(* CODESYS project GlobalConstants.export

Project tree, tasks and I/O mapping:
  GlobalConstants/
    Inficon/
      CommandID/
        global variables InficonHCommandID
        global variables InficonQCCommandID
        global variables InficonQGCommandID
        global variables InficonQMCommandID
        global variables InficonQSCommandID
        global variables InficonRGCommandID
        global variables InficonRLCommandID
        global variables InficonSGCommandID
        global variables InficonSLCommandID
        global variables InficonSSCommandID
      global variables InficonCommand
      global variables InficonQUSubgroup
      global variables InficonResponceErrorCode
      global variables InficonRSSubgroup
    global variables Constants
    global variables IPS_COMMAND
*)

// GlobalConstants/Constants
{attribute 'qualified_only'}
//{attribute 'conditionalshow'}
//{attribute 'conditionalshow' := 'SomeText'}
//{attribute 'hide'}
VAR_GLOBAL CONSTANT
	gc_iDummy : INT := 42; /// This is a dummy global constant variable
END_VAR

// GlobalConstants/IPS_COMMAND
{attribute 'qualified_only'}
VAR_GLOBAL CONSTANT
	START_PERMIT:	UINT:=101;
	START:			UINT:=1;
	STOP:			UINT:=2;
	RESET_ERROR:	UINT:=3;
	
END_VAR

// GlobalConstants/Inficon/InficonCommand
{attribute 'qualified_only'}
(*Основные командные группы.
Команда формируется по следующему шаблону COMMAND_GROUP[SUB GROUP][COMMAND ID](Parameter...Parameter)*)
VAR_GLOBAL CONSTANT
	Hello:BYTE:=STRING_TO_BYTE('H');
	Query:BYTE:=STRING_TO_BYTE('Q');
	RemoteAction:BYTE:=STRING_TO_BYTE('R');
	Status:BYTE:=STRING_TO_BYTE('S');
	Update:BYTE:=STRING_TO_BYTE('U');
	
END_VAR

// GlobalConstants/Inficon/InficonQUSubgroup
{attribute 'qualified_only'}
(*Subcommand for command 'Query' and 'Update's*)
VAR_GLOBAL CONSTANT
	Source:			BYTE:=STRING_TO_BYTE('C');
	General:		BYTE:=STRING_TO_BYTE('G');
	InputName: 		BYTE:=STRING_TO_BYTE('I');
	Logic:			BYTE:=STRING_TO_BYTE('L');
	Material:		BYTE:=STRING_TO_BYTE('M');
	MaterialName:	BYTE:=STRING_TO_BYTE('N');
	OutputName:		BYTE:=STRING_TO_BYTE('O');
	Process:		BYTE:=STRING_TO_BYTE('P');
	Sensor:			BYTE:=STRING_TO_BYTE('S');
	TypeOfOutput:	BYTE:=STRING_TO_BYTE('T');
	UserMessage:	BYTE:=STRING_TO_BYTE('V');
END_VAR

// GlobalConstants/Inficon/InficonResponceErrorCode
{attribute 'qualified_only'}
VAR_GLOBAL CONSTANT
	IllegalCommand:					BYTE:=STRING_TO_BYTE('A');
	IllegalParametervalue:			BYTE:=STRING_TO_BYTE('B');
	InvalidChecksum:				BYTE:=STRING_TO_BYTE('C');
	IllegalID:						BYTE:=STRING_TO_BYTE('D');
	DataNotAvailable:				BYTE:=STRING_TO_BYTE('E');
	IllegalFormat:					BYTE:=STRING_TO_BYTE('F');
	CannotDoNow:					BYTE:=STRING_TO_BYTE('F');
	InvalidMessage:					BYTE:=STRING_TO_BYTE('I');
	LengthError:					BYTE:=STRING_TO_BYTE('L');
	TooManyCommands:				BYTE:=STRING_TO_BYTE('M');
	ResponceLengthLarge:			BYTE:=STRING_TO_BYTE('O');
	ProiorCommandFailed:			BYTE:=STRING_TO_BYTE('P');
END_VAR

// GlobalConstants/Inficon/InficonRSSubgroup
{attribute 'qualified_only'}
VAR_GLOBAL CONSTANT
	General:	BYTE:=STRING_TO_BYTE('G');
 	Material:	BYTE:=STRING_TO_BYTE('L');
	Sensor:		BYTE:=STRING_TO_BYTE('S');
END_VAR

// GlobalConstants/Inficon/CommandID/InficonHCommandID
{attribute 'qualified_only'}
VAR_GLOBAL
	NameAndVersion: 	BYTE:=16#01;
	VersionNumbers:		BYTE:=16#02;
	FirmawareVersion: 	BYTE:=16#03;
END_VAR

// GlobalConstants/Inficon/CommandID/InficonQCCommandID
{attribute 'qualified_only'}
VAR_GLOBAL CONSTANT
	DACOutput: 			BYTE:=16#01;
	ShutterOutput:		BYTE:=16#02;
	NumberOfCrucibles:	BYTE:=16#03;
	CrucibleOutput:		BYTE:=16#04;
	TurretFeedback:		BYTE:=16#05;
	TurretInput:		BYTE:=16#06;
	TurretDelay:		BYTE:=16#07;
END_VAR

// GlobalConstants/Inficon/CommandID/InficonQGCommandID
{attribute 'qualified_only'}
VAR_GLOBAL CONSTANT
	ThinknessEq1:		BYTE:=16#09;
	ThinknessEq2:		BYTE:=16#0A;
	ThinknessEq3:		BYTE:=16#0B;
	Test:				BYTE:=16#0C;
	TimeCompressed:		BYTE:=16#0D;//10x time acceleration
	AdvancedTest:		BYTE:=16#0E;//Crystal Fails Active
	AudioFeedback:		BYTE:=16#0F;
	LCDDimmerTime:		BYTE:=16#10;
	DateFormat:			BYTE:=16#11;
	USBDatalogFormat:	BYTE:=16#12;
	DatalogXtalInfo:	BYTE:=16#13;
	GraphScale:			BYTE:=16#14;
	GraphScaleRate:		BYTE:=16#15;
	RS232Baudrate:		BYTE:=16#16;
	RS232Protocol:		BYTE:=16#17;
	DAC1Scale:			BYTE:=16#18;
	DAC2Scale:			BYTE:=16#19;
	DAC3Scale:			BYTE:=16#1A;
	DAC4Scale:			BYTE:=16#1B;
	DAC5Scale:			BYTE:=16#1C;
	DAC6Scale:			BYTE:=16#1D;
	DAC7Scale:			BYTE:=16#1E;
	DAC8Scale:			BYTE:=16#1F;
	DAC9Scale:			BYTE:=16#20;
	DAC10Scale:			BYTE:=16#21;
	DAC11Scale:			BYTE:=16#22;
	DAC12Scale:			BYTE:=16#23;
	DAC1Polarity:		BYTE:=16#24;
	DAC2Polarity:		BYTE:=16#25;
	DAC3Polarity:		BYTE:=16#26;
	DAC4Polarity:		BYTE:=16#27;
	DAC5Polarity:		BYTE:=16#28;
	DAC6Polarity:		BYTE:=16#29;
	DAC7Polarity:		BYTE:=16#2A;
	DAC8Polarity:		BYTE:=16#2B;
	DAC9Polarity:		BYTE:=16#2C;
	DAC10Polarity:		BYTE:=16#2D;
	DAC11Polarity:		BYTE:=16#2E;
	DAC12Polarity:		BYTE:=16#2F;
	Channel1GraphScale:	BYTE:=16#31;
	Channel2GraphScale:	BYTE:=16#32;
	Channel3GraphScale:	BYTE:=16#33;
	Channel4GraphScale:	BYTE:=16#34;
	Channel5GraphScale:	BYTE:=16#35;
	Channel6GraphScale:	BYTE:=16#36;
	
	
END_VAR

// GlobalConstants/Inficon/CommandID/InficonQMCommandID
{attribute 'qualified_only'}
VAR_GLOBAL CONSTANT
	Density:			BYTE:=16#01;
	ZRation:			BYTE:=16#02;
	MasterTooling:		BYTE:=16#03;
	ControlLoop:		BYTE:=16#04;
	ProcessGain:		BYTE:=16#05;
	TimeConstant:		BYTE:=16#06;
	DeadTime:			BYTE:=16#07;
	MaximumPower:		BYTE:=16#09;
	MinimumPower:		BYTE:=16#0A;
	MaxPowerOption:		BYTE:=16#0B;
	PreCondSoakPower:	BYTE:=16#0C;
	PreCondRiseTime:	BYTE:=16#0D;
	PreCondSoakTime:	BYTE:=16#0E;
	SoakPower1:			BYTE:=16#0F;
	RiseTime1:			BYTE:=16#10;
	SoakTime1:			BYTE:=16#11;
	SoakPower2:			BYTE:=16#12;
	RiseTime2:			BYTE:=16#13;
	SoakTime:			BYTE:=16#14;
	AutoSoak2:			BYTE:=16#15;
	DepAfterPreDep:		BYTE:=16#16;
	DelayOption:		BYTE:=16#17;
	ControlDelayTime:	BYTE:=16#18;
	ShutterDelayAccur:	BYTE:=16#19;
	FeedPower:			BYTE:=16#1C;
	FeedRampTime:		BYTE:=16#1D;
	FeedTime:			BYTE:=16#1E;
	IdlePower:			BYTE:=16#20;
	Rate:				BYTE:=16#21;
	TimeLimit:			BYTE:=16#22;
	RateFilterTime:		BYTE:=16#23;
	TimePowerAvg:		BYTE:=16#24;
	IonAssitDeposite:	BYTE:=16#25;
	OnFinalThinckness:	BYTE:=16#26;
	Ramp1Rate:			BYTE:=16#27;
	StartRamp1:			BYTE:=16#28;
	Ramp1Time:			BYTE:=16#29;
	Ramp2Rate:			BYTE:=16#2A;
	StartRamp2:			BYTE:=16#2B;
	Ramp2Time:			BYTE:=16#2C;
	RateWatvherOption:	BYTE:=16#2D;
	RateWatcherTime:	BYTE:=16#2E;
	RateWatcherAccuracy:BYTE:=16#2F;
	FailureAction:		BYTE:=16#73;
	CrystalTwoTooling:	BYTE:=16#74;
	XtalPositionFirst:	BYTE:=16#75;
	XtalPositionLast:	BYTE:=16#76;
	QaulityPercent:		BYTE:=16#79;
	QualityCounts:		BYTE:=16#7A;
	StabilitySingle:	BYTE:=16#7B;
	StabilityTotal:		BYTE:=16#7C;
	RecorderOutput:		BYTE:=16#7D;
	RecorderFunction:	BYTE:=16#7E;
	RecorderRange:		BYTE:=16#7F;
	
	
	
END_VAR

// GlobalConstants/Inficon/CommandID/InficonQSCommandID
{attribute 'qualified_only'}
VAR_GLOBAL CONSTANT
	ShutterOut:			BYTE:=16#01;
	SensorType:			BYTE:=16#02;
	SitchOut:			BYTE:=16#03;
	AutoZ:				BYTE:=16#04;
	NumberOfPosition:	BYTE:=16#05;
	NumberOfPulse:		BYTE:=16#06;
	PulseOn:			BYTE:=16#07;
	PulseOff:			BYTE:=16#08;
	RecorderOutput:		BYTE:=16#09;
	RecorderFunction:	BYTE:=16#0A;
	RecorderRange:		BYTE:=16#0B;
	
END_VAR

// GlobalConstants/Inficon/CommandID/InficonRGCommandID
{attribute 'qualified_only'}
VAR_GLOBAL CONSTANT
	StopAll:						BYTE:=16#01;
	ResetAll:						BYTE:=16#02;
	RemoteLockOn:					BYTE:=16#03;
	RemoteLockOff:					BYTE:=16#04;
	SetLogicStatement:				BYTE:=16#05;
	ClearLogicStatement:			BYTE:=16#06;
	CrystalFailInhibitOn:			BYTE:=16#07;
	CrystalFailInhibitOff:			BYTE:=16#08;
	SetDate:						BYTE:=16#09;
	SetTime:						BYTE:=16#0A;
	ZeroCounter:					BYTE:=16#0B;
	ZeroTimer:						BYTE:=16#0C;
	StartTimer:						BYTE:=16#0D;
	ClockHoldOn:					BYTE:=16#0F;
	ClockHoldOff:					BYTE:=16#10;
	UserMessageOn:					BYTE:=16#11;
	UserMessageOff:					BYTE:=16#12;
	SoakHold1On:					BYTE:=16#13;
	SoakHold1Off:					BYTE:=16#14;
	SoakHold2On:					BYTE:=16#15;
	SoakHold2Off:					BYTE:=16#16;
	SwitchSensor:					BYTE:=16#17;
	ClearFailedCrystalsX:			BYTE:=16#18;
	RotateHeadX:					BYTE:=16#1A;
	DefaultAllParameters:			BYTE:=16#1B;
	SoakHoldPreConOn:				BYTE:=16#1D;
	SoakHoldPrecomOff:				BYTE:=16#1E;
	StartInhibitOn:					BYTE:=16#1F;
	StartIngibitOff:				BYTE:=16#20;
	RateWatcherSamplingInhibitOn:	BYTE:=16#21;
	RateWatcherSamplingInhibitOff:	BYTE:=16#22;
	WatcherSamplingInitiateOn:		BYTE:=16#23;
	WatcherSamplingInitiateOff:		BYTE:=16#24;
	ClearQAndSCountsForSensore:		BYTE:=16#25;
	NameMaterial:					BYTE:=16#26;
	
END_VAR

// GlobalConstants/Inficon/CommandID/InficonRLCommandID
{attribute 'qualified_only'}
VAR_GLOBAL CONSTANT
	StopMaterial:			BYTE:=16#00;
	ZeroThickness:			BYTE:=16#01;
	StartDeposit:			BYTE:=16#02;
	GoToNonDepositControl:	BYTE:=16#03;
	GoToPostDeposit:		BYTE:=16#04;
	ContinueDeposit:		BYTE:=16#05;
	GoToManual:				BYTE:=16#06;
	SetPowerlevel:			BYTE:=16#07;
	OpenSourceShutter:		BYTE:=16#08;
	CloseSourceShutter:		BYTE:=16#09;
	SetAverageRate:			BYTE:=16#0A;
	Start:					BYTE:=16#0B;
	ResetMaterial:			BYTE:=16#0C;
	
END_VAR

// GlobalConstants/Inficon/CommandID/InficonSGCommandID
{attribute 'qualified_only'}
VAR_GLOBAL CONSTANT
	OutputStatus: 				BYTE:=16#03; //Responce - 5 bytes. Каждый бит репрезентует OUTPUT
	InputStatus:				BYTE:=16#04; //Responce - 4 bytes
	LogicStatementStatus:		BYTE:=16#05; //Responce - 13 byte
	StatusMessage:				BYTE:=16#06; //Responce - 8 bytes
	StatusMessageDesignators:	BYTE:=16#07;
	TrancientMessages:			BYTE:=16#09; // Responce - 1 bytes
	SensorStatus:				BYTE:=16#0A;
	TimerStatus:				BYTE:=16#0B;
	TimerValue:					BYTE:=16#0C;
	CounterValue:				BYTE:=16#0D;
	ThicknessSum:				BYTE:=16#0E;
	GetDate:					BYTE:=16#0F;
	GetTime:					BYTE:=16#10;
	SystemConfuguration:		BYTE:=16#11;
	
	
END_VAR

// GlobalConstants/Inficon/CommandID/InficonSLCommandID
{attribute 'qualified_only'}
VAR_GLOBAL CONSTANT
	FilteredRate:			BYTE:=16#01;
	DisplayRate:			BYTE:=16#02;
	SourcePowerOutput:		BYTE:=16#03;
	Thickness:				BYTE:=16#04;
	State:					BYTE:=16#05;
	StateTime:				BYTE:=16#06;
	ActiveSensors:			BYTE:=16#07;
	PowerSourceNumber:		BYTE:=16#08;
	AccumulatedLayerTime:	BYTE:=16#09;
	DepositAverageRate:		BYTE:=16#0A;
	DepositAveragePower:	BYTE:=16#0B;
	RawRate:				BYTE:=16#0C;
	OneMinuteAvgForRatePwr:	BYTE:=16#0D;
	RateDeviation:			BYTE:=16#0E;
	StateBeforeStop:		BYTE:=16#0F;
	DataLog:				BYTE:=16#10;
	DataLogwithXtalHistory:	BYTE:=16#11;
	CauseOfStop:			BYTE:=16#12;		
END_VAR

// GlobalConstants/Inficon/CommandID/InficonSSCommandID
{attribute 'qualified_only'}
VAR_GLOBAL CONSTANT
	CrystalLife:		BYTE:=16#00;
	CrystalsRemaning:	BYTE:=16#01;
	CrystalPosition:	BYTE:=16#02;
	SensorStatus:		BYTE:=16#03;
	FundamentalFreq:	BYTE:=16#04;
	FundamentalActivity:BYTE:=16#05;
	CurrentZRation:		BYTE:=16#06;
	AnharmonicFreq:		BYTE:=16#07;
	AnharmonicActivity:	BYTE:=16#08;
	NewCrtystaFreq:		BYTE:=16#09;
	LCQValue:			BYTE:=16#0A;
	SensorThickness:	BYTE:=16#0C;
	
END_VAR
